TYPE (* EtherCAT device revision number from ESI Type/@RevisionNo *)
  (* Standard: 61499-1; Description: Copyright (c) 2026 Sichuan Qunyuan Technology Co., Ltd. This program and the accompanying materials are made available under the terms of the Eclipse Public License 2.0 which is available at https://www.eclipse.org/legal/epl-2.0/ SPDX-License-Identifier: EPL-2.0 *)
  (* Version 1.0, 2026-08-10, Zijun Tang, initial API and implementation *)
  PACKAGE eclipse4diac::io::ethercat;
  {SET_ATTRIBUTE(TARGET, (IInterfaceElement:=FALSE,SubApp:=FALSE,FBType:=TRUE,Application:=FALSE,Connection:=FALSE,FB:=FALSE,DataType:=FALSE))}
  RevisionNo : STRING := ''; (* EtherCAT device revision number *)
END_TYPE
